(* CODESYS project BProjPLS.export

Project tree, tasks and I/O mapping:
  application Application
    libraries: Util, * (System); WagoAppBuilding, 1.0.2.5 (WAGO); WagoSolMTP, 2.7.0.0 (WAGO); WagoAppMath, 1.1.1.2 (WAGO); WagoAppRTU, 1.2.13.1 (WAGO)
    task PLC_Task (cyclic, interval t#50ms, priority 15) calls PLC_PRG
    task TrendRecordingTask (cyclic, interval 100 ms, priority 15) calls VisuTrendStorageAccess.GlobalInstances.g_TrendRecordingManager.CyclicCall
    global variables GVL
    global variables LVL
    program Binary [ST]
    program Control_System_Analog [ST]
    program Controller [ST]
    program Engine_Control [FBD]: AzimuthThrusters_1, AzimuthThrusters_2, SideThrusters
    program PLC_PRG [ST]
    program Search_Lights [FBD]
    program Tank_Control [FBD]: DieselTank_1, DieselTank_2
    function block Tank_Simulation [FBD]
    program Tempered_Tank [FBD]
    Symbols
  text list GlobalTextList
*)

// Application/GVL
{attribute 'qualified_only'}
VAR_GLOBAL
 	


// Auto pilot
AutoPilot: BOOL; 
iActualDir:INT;
iDestination:INT;
iDirection:INT;
rSTW:REAL;
rCurrent:REAL;
iDepth:INT;
iCurrentDir:INT;




// Main Thrusters
AzimuthPort_Effect: REAL; 
AzimuthPort_Temp: REAL;
AzimuthPort_Angle: REAL;
AzimuthPort_OilPressure: REAL; 

AzimuthStarboard_Effect: REAL; 
AzimuthStarboard_Temp: REAL;
AzimuthStarboard_Angle: REAL;
AzimuthStarboard_OilPressure: REAL; 

// Side Thrusters 
BowThruster_Effect: REAL;
BowThruster_Temp: REAL;
AftThruster_Effect: REAL;
AftThruster_Temp: REAL;

// Diesel Tank
rPump_Tank1: REAL;
rPump_Reserve1: REAL;
Level_Tank1: REAL;
Level_Reserve1: REAL;
Temperature_Tank1: REAL;
Temperature_Reserve1: REAL;

rPump_Tank2: REAL; 
rPump_Reserve2: REAL;
Level_Tank2: REAL;
Level_Reserve2: REAL;
Temperature_Tank2: REAL;
Temperature_Reserve2: REAL;

// Tempered Tank
TemperedTank1_Level:REAL;
TemperedTank1_Temp:REAL;
TemperedTank1_Heat:BOOL;
TemperedTank1_PumpEffect:INT;
TemperedTank1_PumpOn:BOOL;
END_VAR

// Application/LVL
{attribute 'qualified_only'}
VAR_GLOBAL
	

//Controller
iBinary: INT; 
xDI1, xDI2,xDI3,xDI4,xDI5,xDI6: BOOL;
rVoltage:REAL;




END_VAR

// Application/PLC_PRG
PROGRAM PLC_PRG
VAR
END_VAR

Binary();
Control_System_Analog();
Tank_Control();
Engine_Control();
Search_Lights();
Tempered_Tank();
Controller();

END_PROGRAM

// Application/Binary
PROGRAM Binary
VAR
//binary value holders
B1,B2,B3,B4,B5,B6: INT;
	

// flip flop ikke i bruk
flip_flop_1, flip_flop_2, flip_flop_3, flip_flop_4, flip_flop_5,
flip_flop_6, flip_flop_7: fbLatchingRelay;


	
END_VAR

// BINERY switches for button DI1 - DI6, when DI8 is OFF. 	
IF NOT DI8 THEN
	IF DI1 THEN
		B1:=1;
	ELSE
		B1:=0;
	END_IF
	IF DI2 THEN
		B2:=2;
	ELSE
		B2:=0;
	END_IF
	IF DI3 THEN
		B3:=4;
	ELSE
		B3:=0;
	END_IF
	IF DI4 THEN
		B4:=8;
	ELSE
		B4:=0;
	END_IF
	IF DI5 THEN
		B5:=16;
	ELSE
		B5:=0;
	END_IF
	IF DI6 THEN
		B6:=32;
	ELSE
		B6:=0;
	END_IF
	
	LVL.iBinary:=B1+B2+B3+B4+B5+B6;
	
END_IF

// BOOLEAN swithces DI1-DI6 when DI8 is ON
IF DI8 THEN
	flip_flop_1(xButton:=DI1);
	flip_flop_2(xButton:=DI2);
	flip_flop_3(xButton:=DI3);
	flip_flop_4(xButton:=DI4);
	flip_flop_5(xButton:=DI5);
	flip_flop_6(xButton:=DI6);
	flip_flop_7(xButton:=DI7);
	
	
	// test1:=flip_flop_1.xSwitchActuator;
	// test2:=flip_flop_2.xSwitchActuator;
	
	GVL.AutoPilot:=flip_flop_1.xSwitchActuator;
	   
	
END_IF

END_PROGRAM

// Application/Control_System_Analog
PROGRAM Control_System_Analog
VAR
	r_xCurrent:REAL;
	r_yCurrent:REAL;
	iCurrentDirRel:INT;
	rWind:REAL:=3.5;
	iWindDir:INT :=35;
	rsTimer:RS;
	tonTimer:ton;
	rRegulator:REAL;
	Course:AnaView;
	Speed:AnaView;
	
	//Depth
	arrDepth:ARRAY[0..20]OF INT :=[53,57,61,70,71,73,69,60,57,58,55,70,75,74,76,70,65,63,62,59,58];
	i:INT:=0;
	tonDepth:ton;
	rsDepth:RS;
	Depth_View:AnaView;
	
    //Autopilot
	rCOG: REAL;
		
	END_VAR

//Styresystem fart + control
tonTimer(IN:=rsTimer.Q1,PT:=T#1S);
rsTimer(SET:=TRUE,RESET1:=tonTimer.Q);
IF DI7 AND NOT DI8 AND LVL.iBinary<=7 THEN
	rRegulator:=TO_REAL(iwRegulator)/3276.0;
	IF LVL.iBinary= 4 AND tonTimer.Q AND NOT GVL.AutoPilot THEN
		GVL.iDirection:=GVL.iDirection+ (TO_INT(rRegulator)-5); // styres likt med controller for thruster angle  
		IF GVL.iDirection>=360 THEN
			GVL.iDirection:=GVL.iDirection-360;
		ELSIF GVL.iDirection<0 THEN
			GVL.iDirection:=GVL.iDirection+360;
		END_IF
		Course(TagName:='Ship Course',V:=GVL.iDirection,VSclMin:=360,VSclMax:=0,VUnit:=eUnits_IEC61158.degree);
	END_IF
	IF LVL.iBinary=1 AND NOT GVL.AutoPilot THEN 
		GVL.rSTW:=rRegulator*1.032-3.0; // kobles opp mot thruster effekt 
		Speed(TagName:='Ship Speed',V:=GVL.rSTW,VSclMin:=-3,VSclMax:=10,VUnit:=eUnits_IEC61158.knot);
	END_IF
	
END_IF




//Dybdemåler   --- en output skal være global 
rsDepth(SET:=TRUE,RESET1:=tonDepth.Q);
tonDepth(IN:=rsDepth.Q1,PT:=T#2S);
IF tonDepth.Q THEN
		GVL.iDepth:=-arrDepth[i];
		Depth_View(TagName:='Depth',V:=GVL.iDepth);
		i:=i+1;
		IF i=20 THEN 
			i:=0;
		END_IF
	END_IF
	
	
	
//Current
iCurrentDirRel:=GVL.iCurrentDir-GVL.iDirection;
IF iCurrentDirRel>=360 THEN
	iCurrentDirRel:=iCurrentDirRel - 360;
ELSIF iCurrentDirRel <0 THEN
	iCurrentDirRel := iCurrentDirRel + 360;
END_IF
IF GVL.rCurrent<GVL.rSTW THEN 
r_xCurrent:=-(cos_r(degreeToAngle(iCurrentDirRel))*GVL.rCurrent);//legg til speed heading
r_yCurrent:=-(sin_r(degreeToAngle(iCurrentDirRel))*GVL.rCurrent); 
rCOG:=sqrt_l(((GVL.rSTW+r_xCurrent)*(GVL.rSTW+r_xCurrent))+((r_yCurrent)*(r_yCurrent)));
GVL.iActualDir:=TO_INT(angleToDegree_r(arcTan(r_yCurrent/(GVL.rSTW+r_xCurrent)))+GVL.iDirection);
IF rCOG=0 THEN GVL.iActualDir:=GVL.iDirection; END_IF
IF GVL.iActualDir<0 THEN GVL.iActualDir:=GVL.iActualDir+360; ELSIF GVL.iActualDir>=360 THEN GVL.iActualDir:=GVL.iActualDir-360; END_IF
	
END_IF





//AutoPilot
IF GVL.AutoPilot THEN
	IF GVL.iDestination=GVL.iActualDir THEN GVL.BowThruster_Effect:=0;GVL.AzimuthPort_Angle:=0;GVL.AzimuthStarboard_Angle:=0;END_IF
	IF GVL.iActualDir<0 THEN GVL.iActualDir:=GVL.iActualDir+360; ELSIF GVL.iActualDir>=360 THEN GVL.iActualDir:=GVL.iActualDir-360; END_IF
	IF GVL.iDirection<0 THEN GVL.iDirection:=GVL.iDirection+360; ELSIF GVL.iDirection>=360 THEN GVL.iDirection:=GVL.iDirection-360; END_IF
	IF GVL.iActualDir>GVL.iDestination AND tontimer.Q THEN
		IF GVL.iActualDir-GVL.iDestination>180 THEN // checks if course minus destination is greater than 180 degrees 
			
			IF GVL.iActualDir-GVL.iDestination>340 THEN // 
				GVL.iDirection:=GVL.iDirection+3;
				GVL.BowThruster_Effect := 100;   //autopilot side and main engines
				GVL.AzimuthPort_Angle := 35;
				GVL.AzimuthStarboard_Angle := 35;
			
			ELSIF GVL.iActualDir-GVL.iDestination>350 THEN
				GVL.iDirection:=GVL.iDirection+2;
				GVL.BowThruster_Effect := 50;   //autopilot side and main engines
				GVL.AzimuthPort_Angle := 20;
				GVL.AzimuthStarboard_Angle := 20;
			ELSE 
				GVL.iDirection:=GVL.iDirection+1;
				GVL.BowThruster_Effect := 25;   //autopilot side and main engines
				GVL.AzimuthPort_Angle := 10;
				GVL.AzimuthStarboard_Angle := 10;
			END_IF
		ELSE
		
			IF GVL.iActualDir-GVL.iDestination>20 THEN
			GVL.iDirection:=GVL.iDirection-3;
			
				GVL.BowThruster_Effect := -100;   //autopilot side and main engines
				GVL.AzimuthPort_Angle := -35;
				GVL.AzimuthStarboard_Angle := -35;
			ELSIF GVL.iDestination-GVL.iActualDir>10 THEN
				GVL.iDirection:=GVL.iDirection-2;
					GVL.BowThruster_Effect := -50;   //autopilot side and main engines
				GVL.AzimuthPort_Angle := -20;
				GVL.AzimuthStarboard_Angle := -20;
			ELSE
				GVL.iDirection:=GVL.iDirection-1;
					GVL.BowThruster_Effect := -25;   //autopilot side and main engines
				GVL.AzimuthPort_Angle := -10;
				GVL.AzimuthStarboard_Angle := -10;
			END_IF
		END_IF
	ELSIF GVL.iDestination>GVL.iActualDir AND tonTimer.Q THEN
		IF GVL.iDestination-GVL.iActualDir>180 THEN
			IF GVL.iDestination-GVL.iActualDir>340 THEN
				GVL.iDirection:=GVL.iDirection-3;
					GVL.BowThruster_Effect := -100;   //autopilot side and main engines
				GVL.AzimuthPort_Angle := -35;
				GVL.AzimuthStarboard_Angle := -35;
			ELSIF GVL.iDestination-GVL.iActualDir>350 THEN
				GVL.iDirection:=GVL.iDirection-2;
					GVL.BowThruster_Effect := -50;   //autopilot side and main engines
				GVL.AzimuthPort_Angle := -20;
				GVL.AzimuthStarboard_Angle := -20;
				
			ELSE
				GVL.iDirection:=GVL.iDirection-1;
					GVL.BowThruster_Effect := -25;   //autopilot side and main engines
				GVL.AzimuthPort_Angle := -10;
				GVL.AzimuthStarboard_Angle := -10;
			END_IF
		ELSE
			IF GVL.iDestination-GVL.iActualDir>20 THEN
				GVL.iDirection:=GVL.iDirection+3;
					GVL.BowThruster_Effect := 100;   //autopilot side and main engines
				GVL.AzimuthPort_Angle := 35;
				GVL.AzimuthStarboard_Angle := 35;
			ELSIF GVL.iDestination-GVL.iActualDir>10 THEN
				GVL.iDirection:=GVL.iDirection+2;
					GVL.BowThruster_Effect := 50;   //autopilot side and main engines
				GVL.AzimuthPort_Angle := 20;
				GVL.AzimuthStarboard_Angle := 20;
			ELSE
				GVL.iDirection:=GVL.iDirection+1;
					GVL.BowThruster_Effect := 25;   //autopilot side and main engines
				GVL.AzimuthPort_Angle := 10;
				GVL.AzimuthStarboard_Angle := 10;
			END_IF
		END_IF
	END_IF
END_IF

END_PROGRAM

// Application/Controller
PROGRAM Controller
VAR
tonTimer: ton; 
rsTimer: rs; 	
rRegulator: REAL;



END_VAR


// Direction
tonTimer(IN:=rsTimer.Q1,PT:=T#1S);
rsTimer(SET:=TRUE,RESET1:=tonTimer.Q);



 
 
 //Scales regulator signal
  rRegulator := FU2POINT(IoConfig_Globals_Mapping.iwRegulator,0,0,32760,100); 
  
 
 IF DI7 AND NOT DI8 AND tonTimer.Q THEN  
     LVL.rVoltage:=TO_REAL(TO_INT(rRegulator))/10;
   
      //Azimuth Thrusters 

     IF LVL.iBinary= 1 THEN 
        GVL.AzimuthPort_Effect:=FU2POINT(LVL.rVoltage,0,-30,10,100);
		GVL.AzimuthStarboard_Effect:=FU2POINT(LVL.rVoltage,0,-30,10,100);
     ELSIF LVL.iBinary= 2 THEN  
           GVL.AzimuthPort_Temp:=FU2POINT(LVL.rVoltage,0,0,10,200);
		   GVL.AzimuthStarboard_Temp:=FU2POINT(LVL.rVoltage,0,0,10,200);
     ELSIF LVL.iBinary= 4 AND NOT GVL.autopilot THEN 
           GVL.AzimuthPort_Angle:=FU2POINT(LVL.rVoltage,0,-35,10,35);
		   GVL.AzimuthStarboard_Angle:=FU2POINT(LVL.rVoltage,0,-35,10,35);
     ELSIF LVL.iBinary= 8 THEN 
           GVL.AzimuthPort_OilPressure:=FU2POINT(LVL.rVoltage,0,0,10,100);
		   GVL.AZIMUTHSTARBOARD_OILPRESSURE:=FU2POINT(LVL.RVOLTAGE,0,0,10,100);

     //Side Thrusters. 
	  ELSIF LVL.iBinary=16+1 AND NOT GVL.autopilot THEN  
            GVL.BowThruster_Effect:=FU2POINT(LVL.rVoltage,0,-100,10,100);
	  ELSIF LVL.iBinary=16+2 
         THEN  GVL.BowThruster_Temp:=FU2POINT(LVL.rVoltage,0,-10,10,200);
   
      ELSIF LVL.iBinary=16+4 
         THEN  GVL.AftThruster_Effect:=FU2POINT(LVL.rVoltage,0,-100,10,100);
      ELSIF LVL.iBinary=16+8
         THEN  GVL.AftThruster_Temp:=FU2POINT(LVL.rVoltage,0,-10,10,200);
		
    // Diesel Tanks 
	ELSIF LVL.iBinary=32+1 THEN
		GVL.Level_Tank1:=FU2POINT(LVL.rVoltage,0,0,10,200);
		GVL.Level_Tank2:=FU2POINT(LVL.rVoltage,0,0,10,200);
	ELSIF LVL.iBinary=32+2 THEN
		GVL.Level_Reserve1:=FU2POINT(LVL.rVoltage,0,0,10,50);
		GVL.Level_Reserve2:=FU2POINT(LVL.rVoltage,0,0,10,50);
	ELSIF LVL.iBinary=32+4 THEN
		GVL.Temperature_Tank1:=FU2POINT(LVL.rVoltage,0,0,10,225);
		GVL.Temperature_Tank2:=FU2POINT(LVL.rVoltage,0,0,10,225);
	ELSIF LVL.iBinary=32+8 THEN
		GVL.Temperature_Reserve1:=FU2POINT(LVL.rVoltage,0,0,10,225);
		GVL.Temperature_Reserve2:=FU2POINT(LVL.rVoltage,0,0,10,225);
	END_IF
			 
   
         
	
END_IF

END_PROGRAM

// Application/Tank_Control
PROGRAM Tank_Control
VAR	
// Variables for fuel controll	
Engine_Effect1: REAL;
Fuelusage1: REAL;

Engine_Effect2: REAL;
Fuelusage2: REAL;


	//Diesel Tank 1

	
	Level_Tank1_Mon: AnaMon :=(VTHLim:=200,VALLim:=1,VWLLim:=10,V:=50);
	Level_Reserve1_Mon: AnaMon :=(VTHLim:=50,VALLim:=1,VWLLim:=5);
	Temperature_Tank1_Mon: AnaMon :=(VAHLim:=200,VWHLim:=100);
	Temperature_Reserve1_Mon: AnaMon :=(VAHLim:=200,VWHLim:=100);



	Pump_Tank1_View: AnaView;
	Pump_Reserve1_View: AnaView;
	

    //Diesel Tank 2


	
	Pump_Tank2_View: AnaView;
	Pump_Reserve2_View: AnaView;
	Level_Tank2_Mon: AnaMon :=(VTHLim:=200,VALLim:=1,VWLLim:=10);
	Level_Reserve2_Mon: AnaMon :=(VTHLim:=50,VALLim:=1,VWLLim:=5);
	Temperature_Tank2_Mon: AnaMon :=(VAHLim:=200,VWHLim:=100);
	Temperature_Reserve2_Mon: AnaMon :=(VAHLim:=200,VWHLim:=100);

	
END_VAR
VAR // added by the converter: edge detectors and wires of the graphical bodies
    _w1, _w2, _w3, _w4 : BOOL;
END_VAR

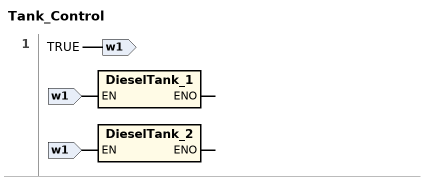
// NETWORK 1
DieselTank_1();
DieselTank_2();

ACTION DieselTank_1:
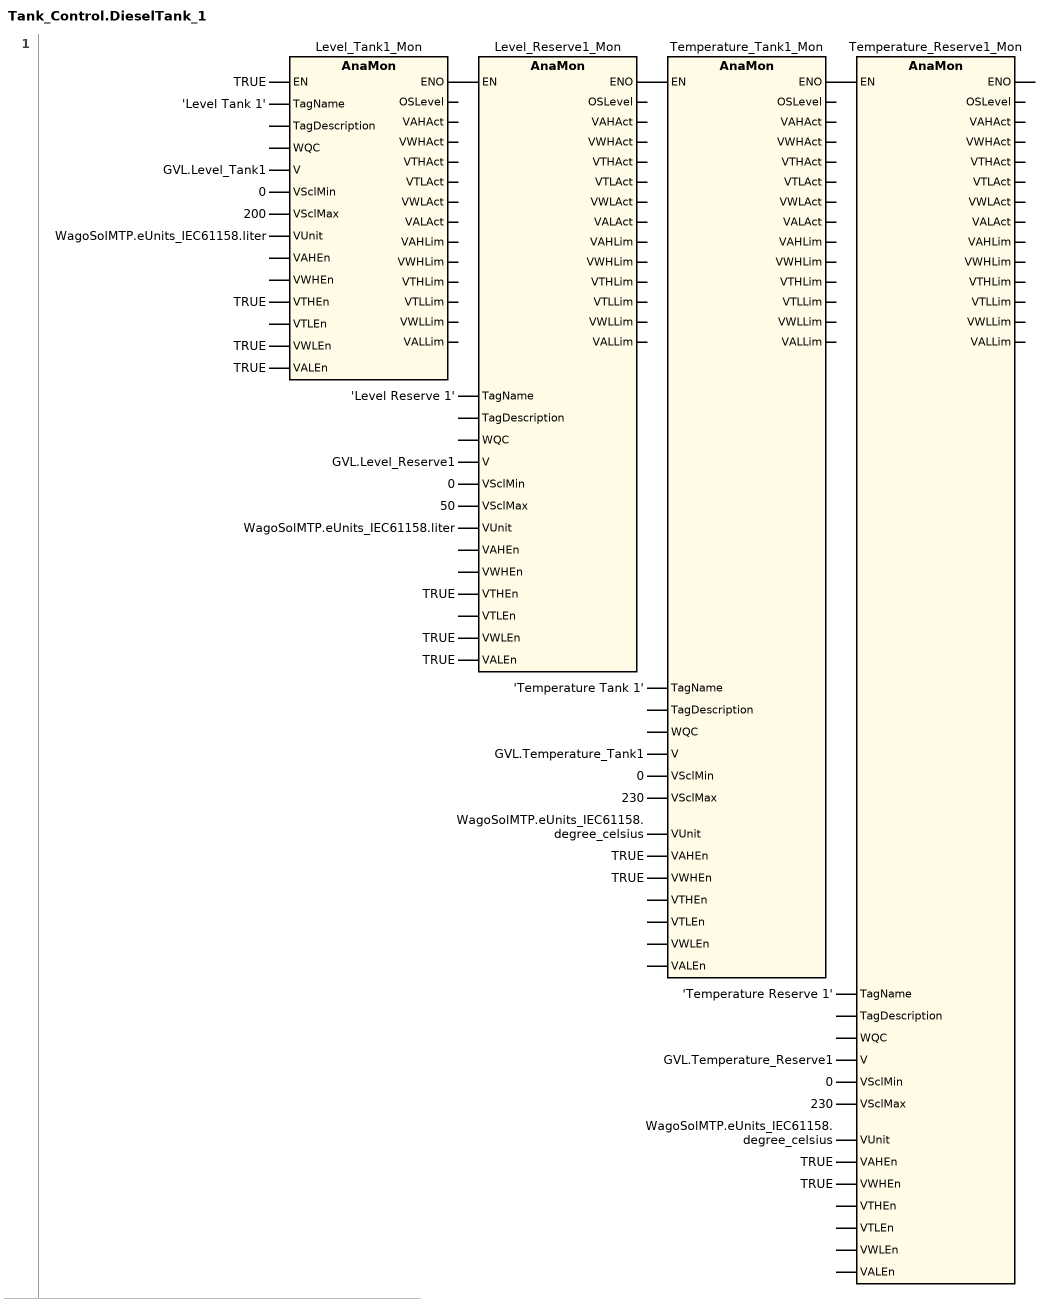
// NETWORK 1
Level_Tank1_Mon(
    TagName := 'Level Tank 1',
    V := GVL.Level_Tank1,
    VSclMin := 0,
    VSclMax := 200,
    VUnit := WagoSolMTP.eUnits_IEC61158.liter,
    VTHEn := TRUE,
    VWLEn := TRUE,
    VALEn := TRUE); // AnaMon
Level_Reserve1_Mon(
    TagName := 'Level Reserve 1',
    V := GVL.Level_Reserve1,
    VSclMin := 0,
    VSclMax := 50,
    VUnit := WagoSolMTP.eUnits_IEC61158.liter,
    VTHEn := TRUE,
    VWLEn := TRUE,
    VALEn := TRUE); // AnaMon
Temperature_Tank1_Mon(
    TagName := 'Temperature Tank 1',
    V := GVL.Temperature_Tank1,
    VSclMin := 0,
    VSclMax := 230,
    VUnit := WagoSolMTP.eUnits_IEC61158.degree_celsius,
    VAHEn := TRUE,
    VWHEn := TRUE); // AnaMon
Temperature_Reserve1_Mon(
    TagName := 'Temperature Reserve 1',
    V := GVL.Temperature_Reserve1,
    VSclMin := 0,
    VSclMax := 230,
    VUnit := WagoSolMTP.eUnits_IEC61158.degree_celsius,
    VAHEn := TRUE,
    VWHEn := TRUE); // AnaMon

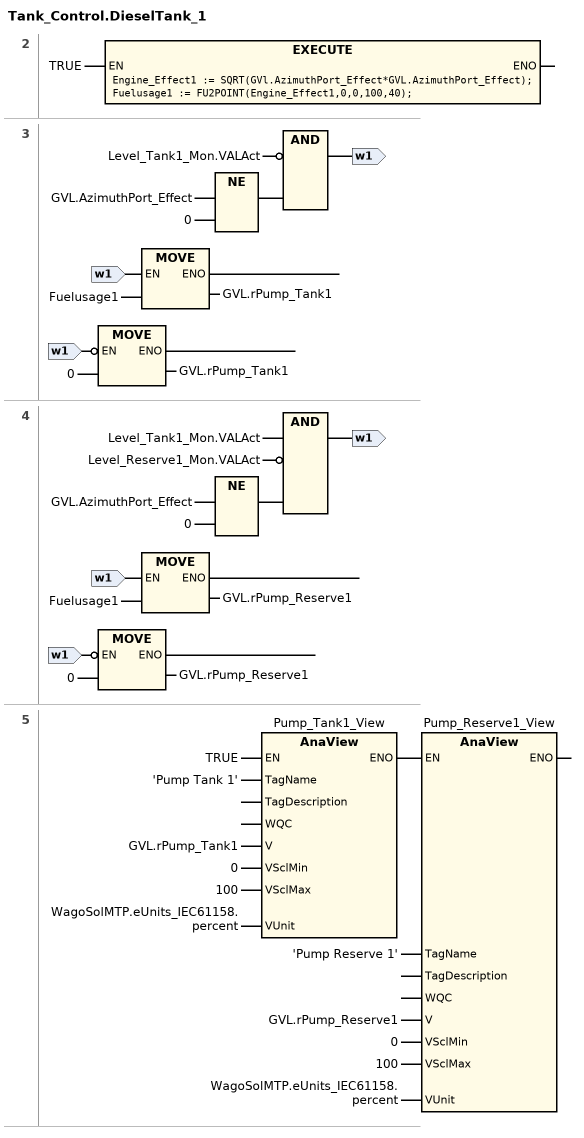
// NETWORK 2
Engine_Effect1 := SQRT(GVl.AzimuthPort_Effect*GVL.AzimuthPort_Effect);
Fuelusage1 := FU2POINT(Engine_Effect1,0,0,100,40);

// NETWORK 3
_w1 := NOT Level_Tank1_Mon.VALAct AND GVL.AzimuthPort_Effect <> 0;
IF _w1 THEN GVL.rPump_Tank1 := Fuelusage1; END_IF
IF NOT _w1 THEN GVL.rPump_Tank1 := 0; END_IF

// NETWORK 4
_w2 := Level_Tank1_Mon.VALAct AND NOT Level_Reserve1_Mon.VALAct AND GVL.AzimuthPort_Effect <> 0;
IF _w2 THEN GVL.rPump_Reserve1 := Fuelusage1; END_IF
IF NOT _w2 THEN GVL.rPump_Reserve1 := 0; END_IF

// NETWORK 5
Pump_Tank1_View(
    TagName := 'Pump Tank 1',
    V := GVL.rPump_Tank1,
    VSclMin := 0,
    VSclMax := 100,
    VUnit := WagoSolMTP.eUnits_IEC61158.percent); // AnaView
Pump_Reserve1_View(
    TagName := 'Pump Reserve 1',
    V := GVL.rPump_Reserve1,
    VSclMin := 0,
    VSclMax := 100,
    VUnit := WagoSolMTP.eUnits_IEC61158.percent); // AnaView
END_ACTION

ACTION DieselTank_2:
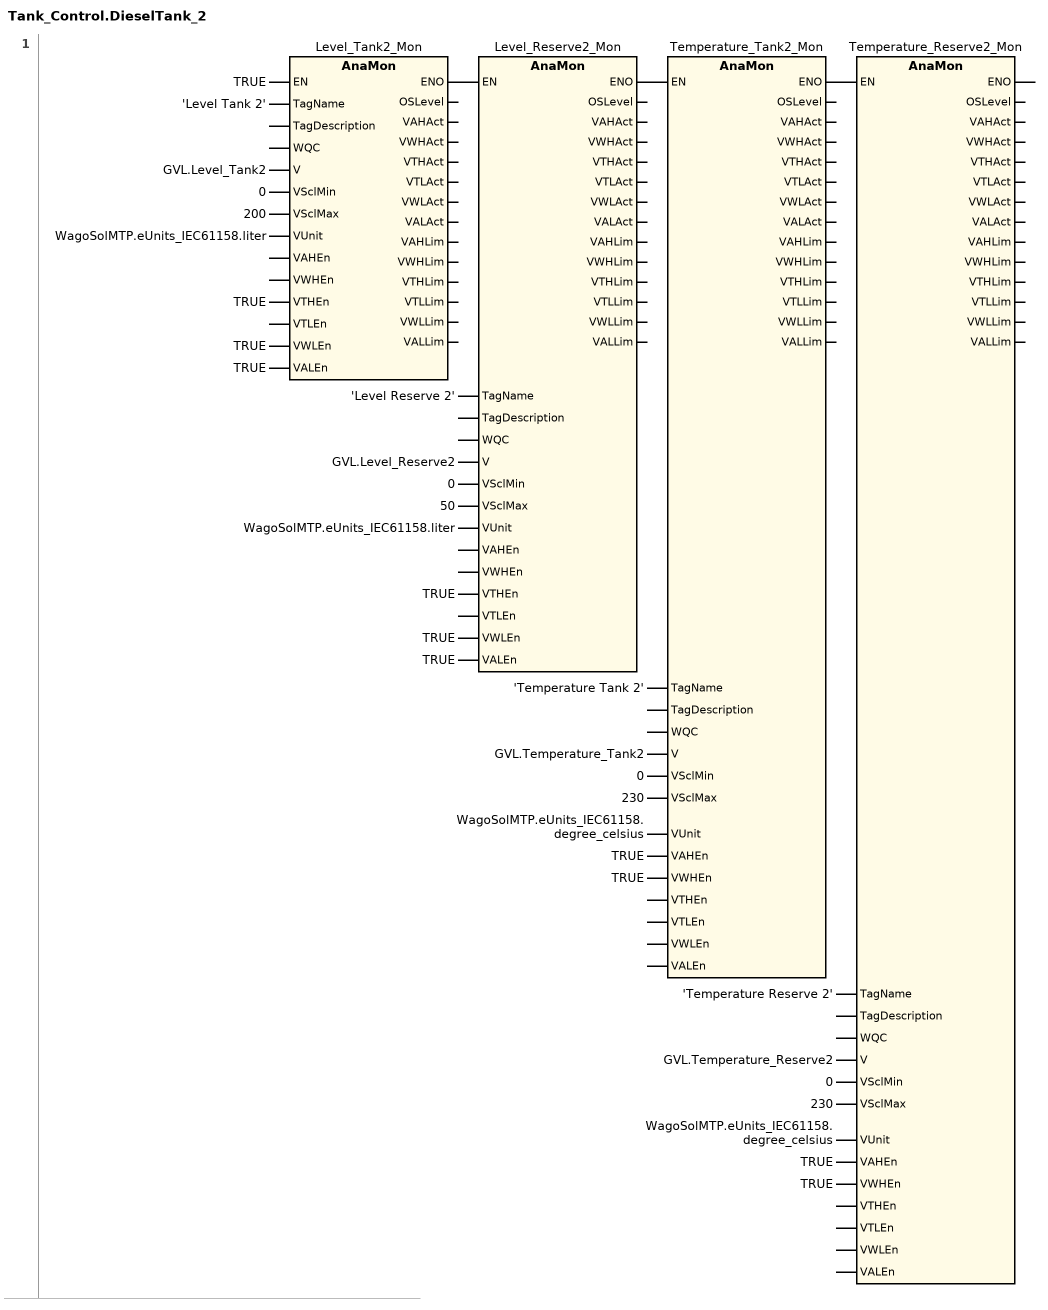
// NETWORK 1
Level_Tank2_Mon(
    TagName := 'Level Tank 2',
    V := GVL.Level_Tank2,
    VSclMin := 0,
    VSclMax := 200,
    VUnit := WagoSolMTP.eUnits_IEC61158.liter,
    VTHEn := TRUE,
    VWLEn := TRUE,
    VALEn := TRUE); // AnaMon
Level_Reserve2_Mon(
    TagName := 'Level Reserve 2',
    V := GVL.Level_Reserve2,
    VSclMin := 0,
    VSclMax := 50,
    VUnit := WagoSolMTP.eUnits_IEC61158.liter,
    VTHEn := TRUE,
    VWLEn := TRUE,
    VALEn := TRUE); // AnaMon
Temperature_Tank2_Mon(
    TagName := 'Temperature Tank 2',
    V := GVL.Temperature_Tank2,
    VSclMin := 0,
    VSclMax := 230,
    VUnit := WagoSolMTP.eUnits_IEC61158.degree_celsius,
    VAHEn := TRUE,
    VWHEn := TRUE); // AnaMon
Temperature_Reserve2_Mon(
    TagName := 'Temperature Reserve 2',
    V := GVL.Temperature_Reserve2,
    VSclMin := 0,
    VSclMax := 230,
    VUnit := WagoSolMTP.eUnits_IEC61158.degree_celsius,
    VAHEn := TRUE,
    VWHEn := TRUE); // AnaMon

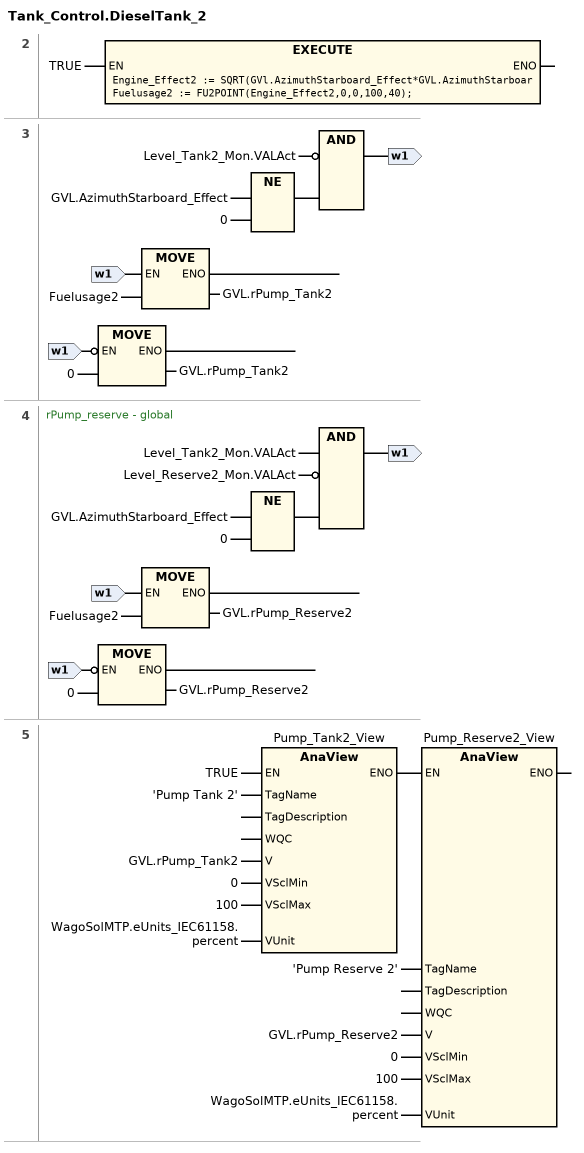
// NETWORK 2
Engine_Effect2 := SQRT(GVl.AzimuthStarboard_Effect*GVL.AzimuthStarboard_Effect);
Fuelusage2 := FU2POINT(Engine_Effect2,0,0,100,40);

// NETWORK 3
_w3 := NOT Level_Tank2_Mon.VALAct AND GVL.AzimuthStarboard_Effect <> 0;
IF _w3 THEN GVL.rPump_Tank2 := Fuelusage2; END_IF
IF NOT _w3 THEN GVL.rPump_Tank2 := 0; END_IF

// NETWORK 4
// rPump_reserve - global
_w4 := Level_Tank2_Mon.VALAct AND NOT Level_Reserve2_Mon.VALAct AND GVL.AzimuthStarboard_Effect <> 0;
IF _w4 THEN GVL.rPump_Reserve2 := Fuelusage2; END_IF
IF NOT _w4 THEN GVL.rPump_Reserve2 := 0; END_IF

// NETWORK 5
Pump_Tank2_View(
    TagName := 'Pump Tank 2',
    V := GVL.rPump_Tank2,
    VSclMin := 0,
    VSclMax := 100,
    VUnit := WagoSolMTP.eUnits_IEC61158.percent); // AnaView
Pump_Reserve2_View(
    TagName := 'Pump Reserve 2',
    V := GVL.rPump_Reserve2,
    VSclMin := 0,
    VSclMax := 100,
    VUnit := WagoSolMTP.eUnits_IEC61158.percent); // AnaView
END_ACTION

END_PROGRAM

// Application/Engine_Control
PROGRAM Engine_Control
VAR


    //AzimuthThruster
   
 
    //Side Thrusters
   
	
	//Thruster 1
	AzimuthPort_Angle_View: AnaView;
	AzimuthPort_OilPressure_View: AnaView;
	
	AzimuthPort_Temp_Mon: AnaMon:= (VAHLim:= 200, VWHLim:= 150, VALLim:=-10);
	AzimuthPort_Effect_Mon: AnaMon:= (VAHLim:= 100, VTHLim:=80, VALLim:= -30);
	
	
	
	//Thruster 2
	AzimuthStarboard_Angle_View: AnaView;
	AzimuthStarboard_OilPressure_View: AnaView;
	
	AzimuthStarboard_Temp_Mon: AnaMon:= (VAHLim:= 200, VWHLim:= 150, VALLim:=-10);
	AzimuthStarboard_Effect_Mon: AnaMon:= (VAHLim:= 100, VTHLim:=80, VALLim:= -30);
	
	
	
	// Bow Thruster 1
    
    BowThruster1_Effect_View: AnaView;
	BowThruster1_Temp_View: AnaView;
    
    BowThruster1_Temp_Mon: AnaMon:= (VAHLim:= 200, VWHLim:= 150, VALLim:=-10);
							
	//Bow Thruster 2
   	BowThruster2_Effect_View: AnaView;
	BowThruster2_Temp_View: AnaView;
	
    BowThruster2_Temp_Mon: AnaMon :=(VAHLim:= 200, VWHLim:= 150, VALLim:=-10);
	
	//AftThruster 2 
	AftThruster_Effect_View: AnaView;
	AftThruster_Temp_View: AnaView;
	
    AftThruster_Temp_Mon: AnaMon := (VAHLim:= 200, VWHLim:= 150, VALLim:=-10);
	
	
	
	
 



END_VAR

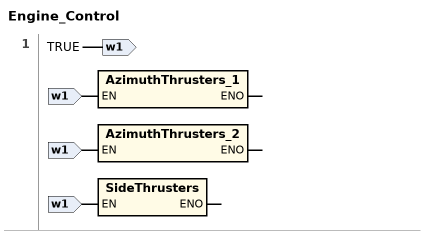
// NETWORK 1
AzimuthThrusters_1();
AzimuthThrusters_2();
SideThrusters();

ACTION AzimuthThrusters_1:
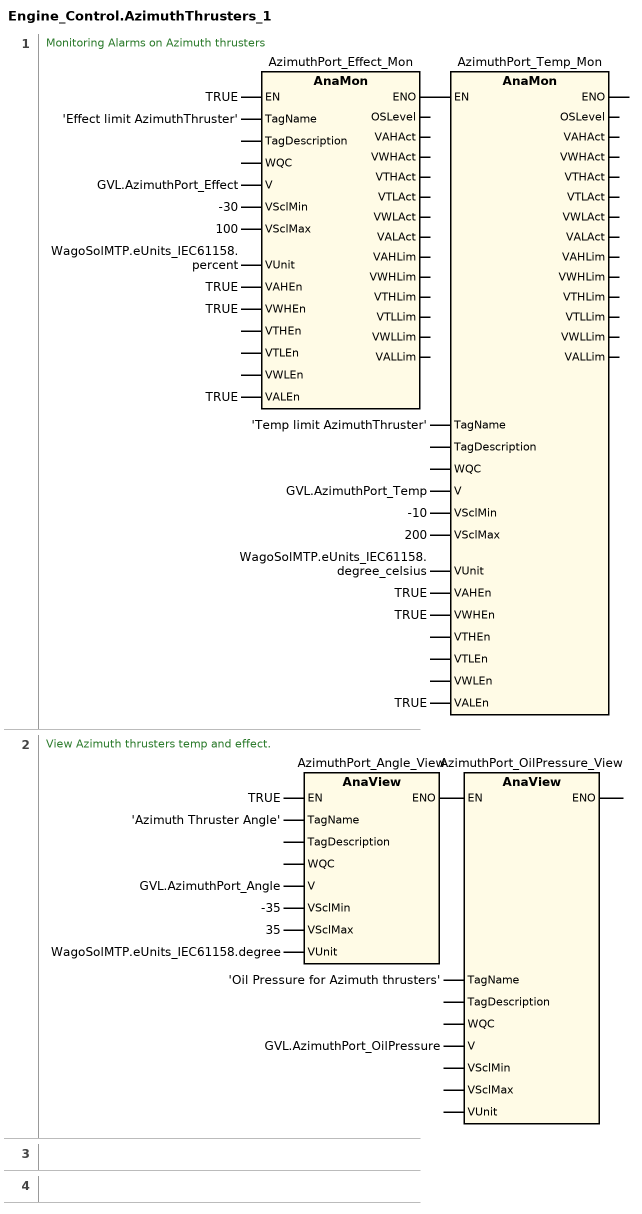
// NETWORK 1
// Monitoring Alarms on Azimuth thrusters
AzimuthPort_Effect_Mon(
    TagName := 'Effect limit AzimuthThruster',
    V := GVL.AzimuthPort_Effect,
    VSclMin := -30,
    VSclMax := 100,
    VUnit := WagoSolMTP.eUnits_IEC61158.percent,
    VAHEn := TRUE,
    VWHEn := TRUE,
    VALEn := TRUE); // AnaMon
AzimuthPort_Temp_Mon(
    TagName := 'Temp limit AzimuthThruster',
    V := GVL.AzimuthPort_Temp,
    VSclMin := -10,
    VSclMax := 200,
    VUnit := WagoSolMTP.eUnits_IEC61158.degree_celsius,
    VAHEn := TRUE,
    VWHEn := TRUE,
    VALEn := TRUE); // AnaMon

// NETWORK 2
// View Azimuth thrusters temp and effect.
AzimuthPort_Angle_View(
    TagName := 'Azimuth Thruster Angle',
    V := GVL.AzimuthPort_Angle,
    VSclMin := -35,
    VSclMax := 35,
    VUnit := WagoSolMTP.eUnits_IEC61158.degree); // AnaView
AzimuthPort_OilPressure_View(TagName := 'Oil Pressure for Azimuth thrusters', V := GVL.AzimuthPort_OilPressure); // AnaView

// NETWORK 3

// NETWORK 4
END_ACTION

ACTION AzimuthThrusters_2:
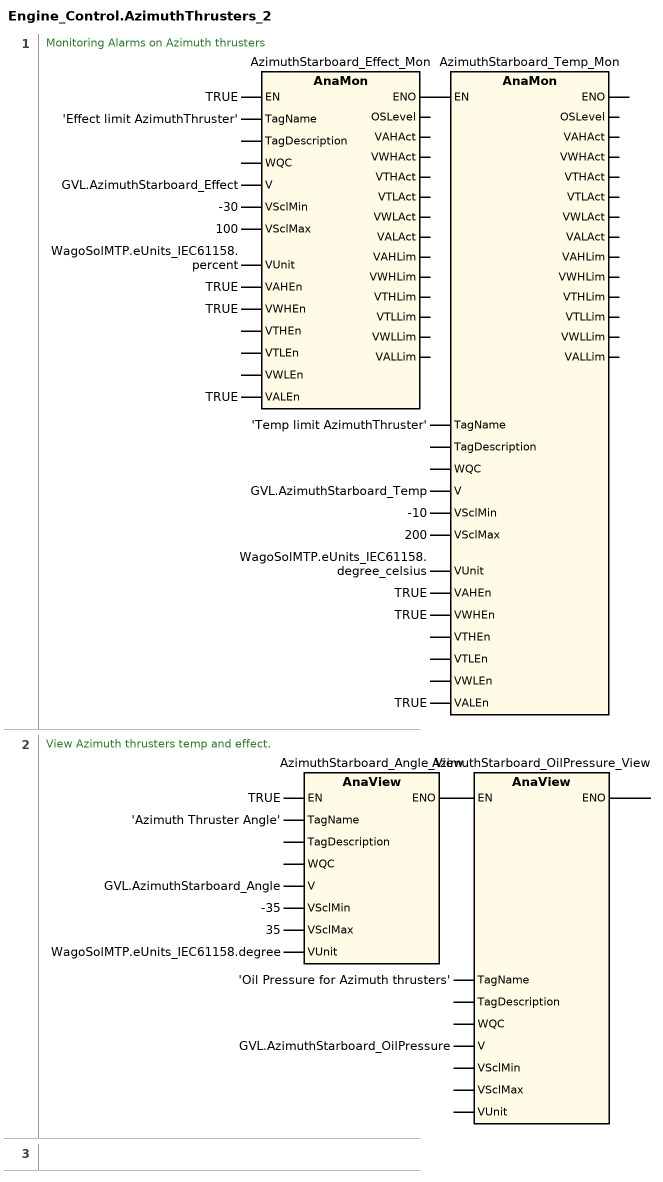
// NETWORK 1
// Monitoring Alarms on Azimuth thrusters
AzimuthStarboard_Effect_Mon(
    TagName := 'Effect limit AzimuthThruster',
    V := GVL.AzimuthStarboard_Effect,
    VSclMin := -30,
    VSclMax := 100,
    VUnit := WagoSolMTP.eUnits_IEC61158.percent,
    VAHEn := TRUE,
    VWHEn := TRUE,
    VALEn := TRUE); // AnaMon
AzimuthStarboard_Temp_Mon(
    TagName := 'Temp limit AzimuthThruster',
    V := GVL.AzimuthStarboard_Temp,
    VSclMin := -10,
    VSclMax := 200,
    VUnit := WagoSolMTP.eUnits_IEC61158.degree_celsius,
    VAHEn := TRUE,
    VWHEn := TRUE,
    VALEn := TRUE); // AnaMon

// NETWORK 2
// View Azimuth thrusters temp and effect.
AzimuthStarboard_Angle_View(
    TagName := 'Azimuth Thruster Angle',
    V := GVL.AzimuthStarboard_Angle,
    VSclMin := -35,
    VSclMax := 35,
    VUnit := WagoSolMTP.eUnits_IEC61158.degree); // AnaView
AzimuthStarboard_OilPressure_View(TagName := 'Oil Pressure for Azimuth thrusters', V := GVL.AzimuthStarboard_OilPressure); // AnaView

// NETWORK 3
END_ACTION

ACTION SideThrusters:
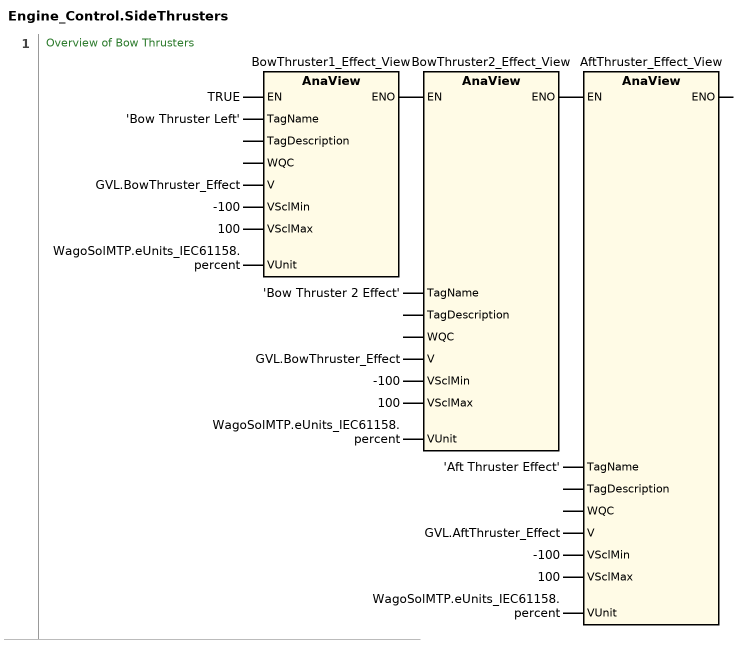
// NETWORK 1
// Overview of Bow Thrusters
BowThruster1_Effect_View(
    TagName := 'Bow Thruster Left',
    V := GVL.BowThruster_Effect,
    VSclMin := -100,
    VSclMax := 100,
    VUnit := WagoSolMTP.eUnits_IEC61158.percent); // AnaView
BowThruster2_Effect_View(
    TagName := 'Bow Thruster 2 Effect',
    V := GVL.BowThruster_Effect,
    VSclMin := -100,
    VSclMax := 100,
    VUnit := WagoSolMTP.eUnits_IEC61158.percent); // AnaView
AftThruster_Effect_View(
    TagName := 'Aft Thruster Effect',
    V := GVL.AftThruster_Effect,
    VSclMin := -100,
    VSclMax := 100,
    VUnit := WagoSolMTP.eUnits_IEC61158.percent); // AnaView

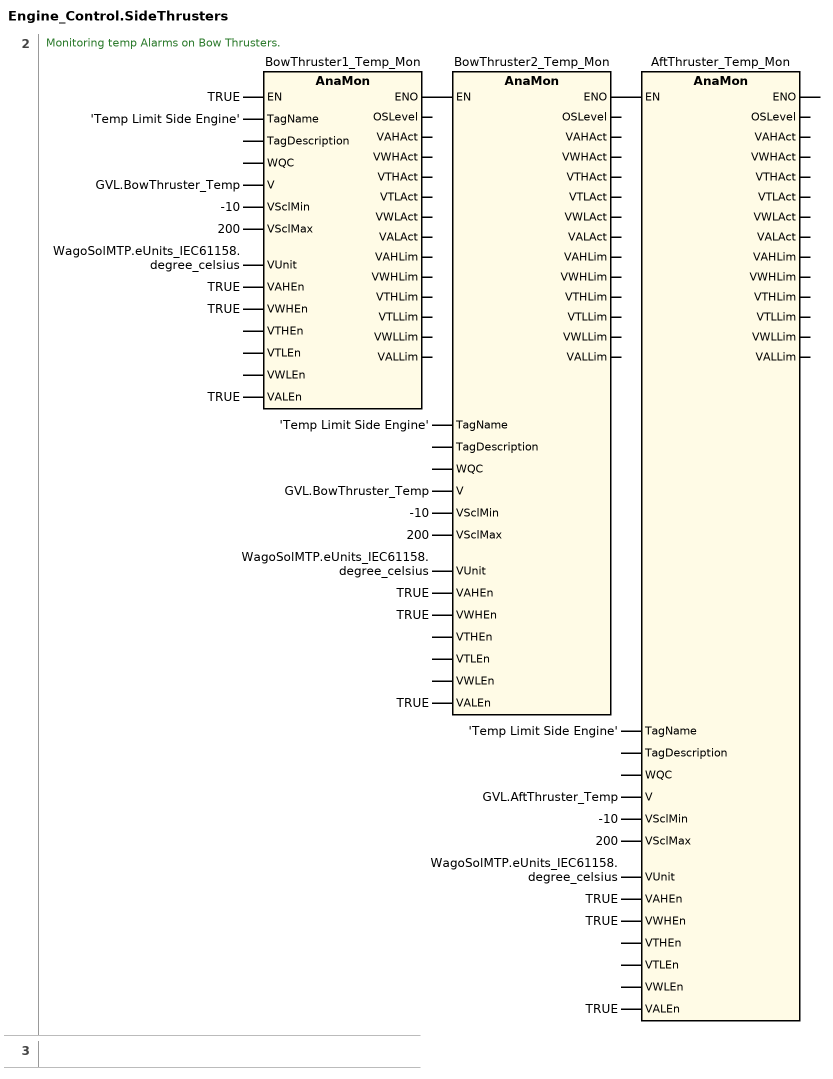
// NETWORK 2
// Monitoring temp Alarms on Bow Thrusters.
BowThruster1_Temp_Mon(
    TagName := 'Temp Limit Side Engine',
    V := GVL.BowThruster_Temp,
    VSclMin := -10,
    VSclMax := 200,
    VUnit := WagoSolMTP.eUnits_IEC61158.degree_celsius,
    VAHEn := TRUE,
    VWHEn := TRUE,
    VALEn := TRUE); // AnaMon
BowThruster2_Temp_Mon(
    TagName := 'Temp Limit Side Engine',
    V := GVL.BowThruster_Temp,
    VSclMin := -10,
    VSclMax := 200,
    VUnit := WagoSolMTP.eUnits_IEC61158.degree_celsius,
    VAHEn := TRUE,
    VWHEn := TRUE,
    VALEn := TRUE); // AnaMon
AftThruster_Temp_Mon(
    TagName := 'Temp Limit Side Engine',
    V := GVL.AftThruster_Temp,
    VSclMin := -10,
    VSclMax := 200,
    VUnit := WagoSolMTP.eUnits_IEC61158.degree_celsius,
    VAHEn := TRUE,
    VWHEn := TRUE,
    VALEn := TRUE); // AnaMon

// NETWORK 3
END_ACTION

END_PROGRAM

// Application/Search_Lights
PROGRAM Search_Lights
VAR
	Search_Light_1: AnaMan;
	Search_Light_2: AnaMan;
	Search_Light_3: AnaMan;
	Search_Light_4: AnaMan;
	Search_Light_5: AnaMan;
	Search_Light_6: AnaMan;
	Search_Light_7: AnaMan;
	Light_Switch_1: BinMan;
	Light_Switch_2: BinMan;
	Light_Switch_3: BinMan;
	Light_Switch_4: BinMan;
	Light_Switch_5: BinMan;
	Light_Switch_6: BinMan;
	Light_Switch_7: BinMan;
END_VAR

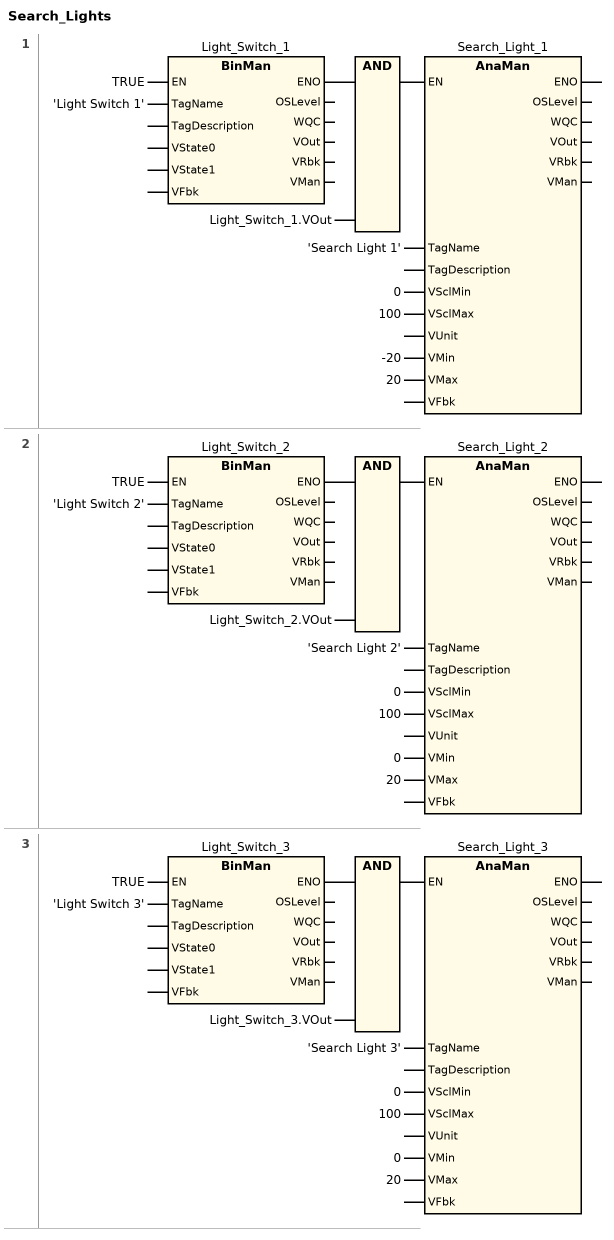
// NETWORK 1
Light_Switch_1(TagName := 'Light Switch 1'); // BinMan
IF TRUE AND Light_Switch_1.VOut THEN
    Search_Light_1(TagName := 'Search Light 1', VSclMin := 0, VSclMax := 100, VMin := -20, VMax := 20); // AnaMan
END_IF

// NETWORK 2
Light_Switch_2(TagName := 'Light Switch 2'); // BinMan
IF TRUE AND Light_Switch_2.VOut THEN
    Search_Light_2(TagName := 'Search Light 2', VSclMin := 0, VSclMax := 100, VMin := 0, VMax := 20); // AnaMan
END_IF

// NETWORK 3
Light_Switch_3(TagName := 'Light Switch 3'); // BinMan
IF TRUE AND Light_Switch_3.VOut THEN
    Search_Light_3(TagName := 'Search Light 3', VSclMin := 0, VSclMax := 100, VMin := 0, VMax := 20); // AnaMan
END_IF

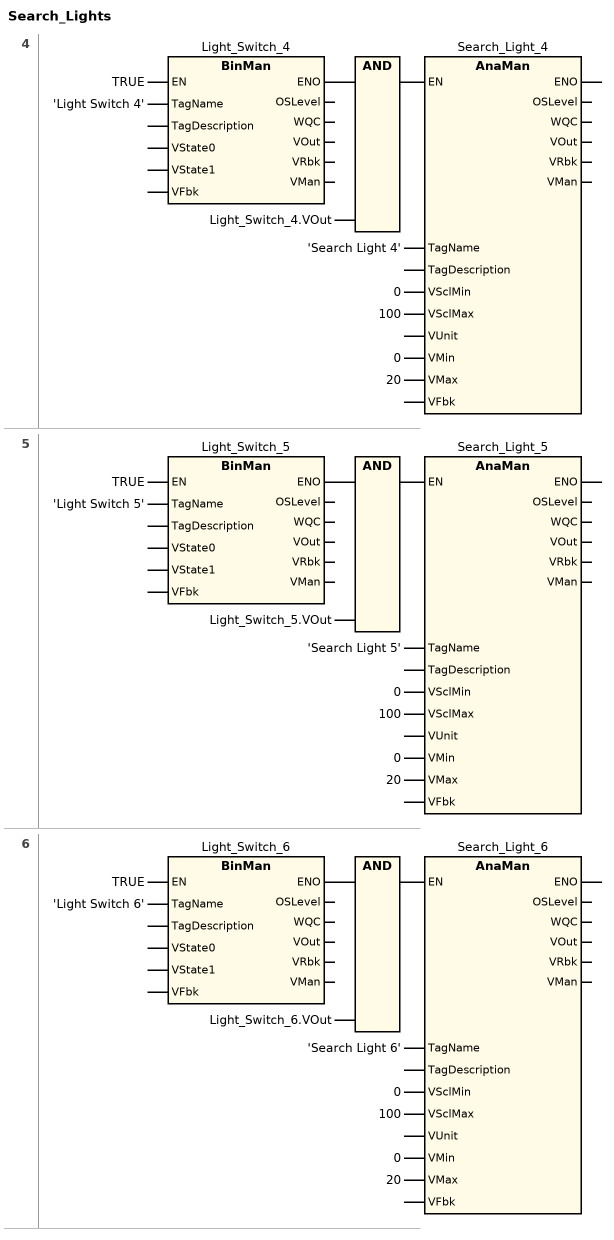
// NETWORK 4
Light_Switch_4(TagName := 'Light Switch 4'); // BinMan
IF TRUE AND Light_Switch_4.VOut THEN
    Search_Light_4(TagName := 'Search Light 4', VSclMin := 0, VSclMax := 100, VMin := 0, VMax := 20); // AnaMan
END_IF

// NETWORK 5
Light_Switch_5(TagName := 'Light Switch 5'); // BinMan
IF TRUE AND Light_Switch_5.VOut THEN
    Search_Light_5(TagName := 'Search Light 5', VSclMin := 0, VSclMax := 100, VMin := 0, VMax := 20); // AnaMan
END_IF

// NETWORK 6
Light_Switch_6(TagName := 'Light Switch 6'); // BinMan
IF TRUE AND Light_Switch_6.VOut THEN
    Search_Light_6(TagName := 'Search Light 6', VSclMin := 0, VSclMax := 100, VMin := 0, VMax := 20); // AnaMan
END_IF

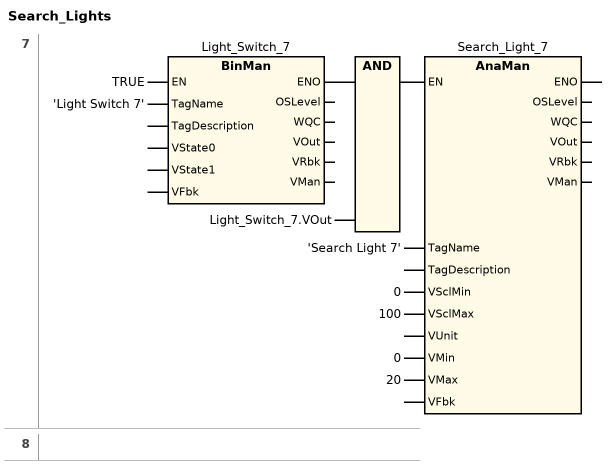
// NETWORK 7
Light_Switch_7(TagName := 'Light Switch 7'); // BinMan
IF TRUE AND Light_Switch_7.VOut THEN
    Search_Light_7(TagName := 'Search Light 7', VSclMin := 0, VSclMax := 100, VMin := 0, VMax := 20); // AnaMan
END_IF

// NETWORK 8

END_PROGRAM

// Application/Tempered_Tank
PROGRAM Tempered_Tank
VAR
	//Tank 1 --- sett global 
	Set_Temp_1: Anaman;
	Tank_Simu_1: Tank_Simulation;
	Tank_Level_1: AnaView;
	Tank_Temp_1: AnaView;
	Tank_Heater_1: binview;

	//Tank 2
	Set_Temp_2: Anaman;
	Tank_Simu_2: Tank_Simulation;
	Tank_Level_2: AnaView;
	Tank_Temp_2: AnaView;
	Tank_Heater_2: binview;

	//Tank 3
	Set_Temp_3: Anaman;
	Tank_Simu_3: Tank_Simulation;
	Tank_Level_3: AnaView;
	Tank_Temp_3: AnaView;
	Tank_Heater_3: binview;

	//Tank 4
	Set_Temp_4: Anaman;
	Tank_Simu_4: Tank_Simulation;
	Tank_Level_4: AnaView;
	Tank_Temp_4: AnaView;
	Tank_Heater_4: binview;
END_VAR

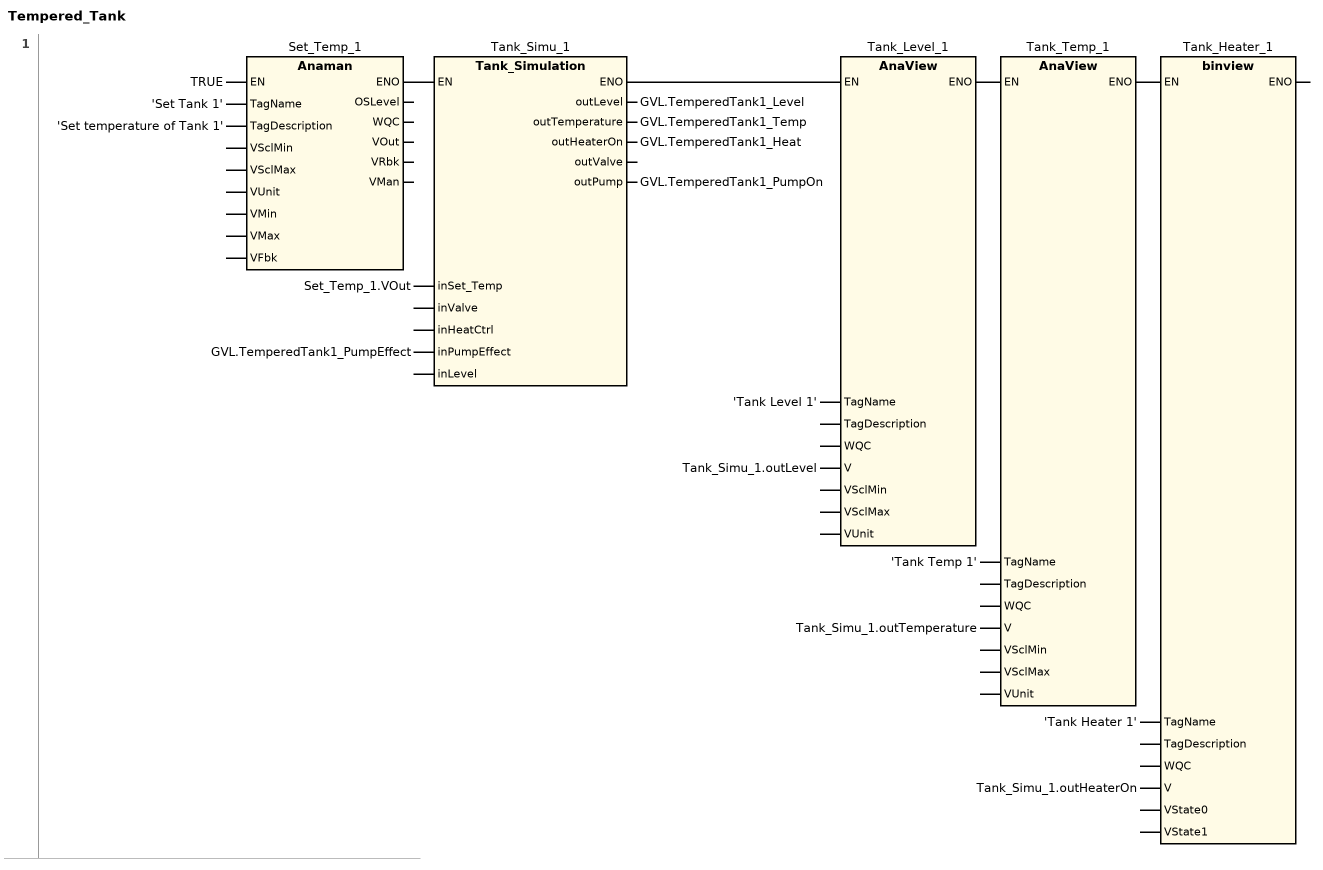
// NETWORK 1
Set_Temp_1(TagName := 'Set Tank 1', TagDescription := 'Set temperature of Tank 1'); // Anaman
Tank_Simu_1(
    inSet_Temp := Set_Temp_1.VOut,
    inPumpEffect := GVL.TemperedTank1_PumpEffect,
    outLevel => GVL.TemperedTank1_Level,
    outTemperature => GVL.TemperedTank1_Temp,
    outHeaterOn => GVL.TemperedTank1_Heat,
    outPump => GVL.TemperedTank1_PumpOn); // Tank_Simulation
Tank_Level_1(TagName := 'Tank Level 1', V := Tank_Simu_1.outLevel); // AnaView
Tank_Temp_1(TagName := 'Tank Temp 1', V := Tank_Simu_1.outTemperature); // AnaView
Tank_Heater_1(TagName := 'Tank Heater 1', V := Tank_Simu_1.outHeaterOn); // binview

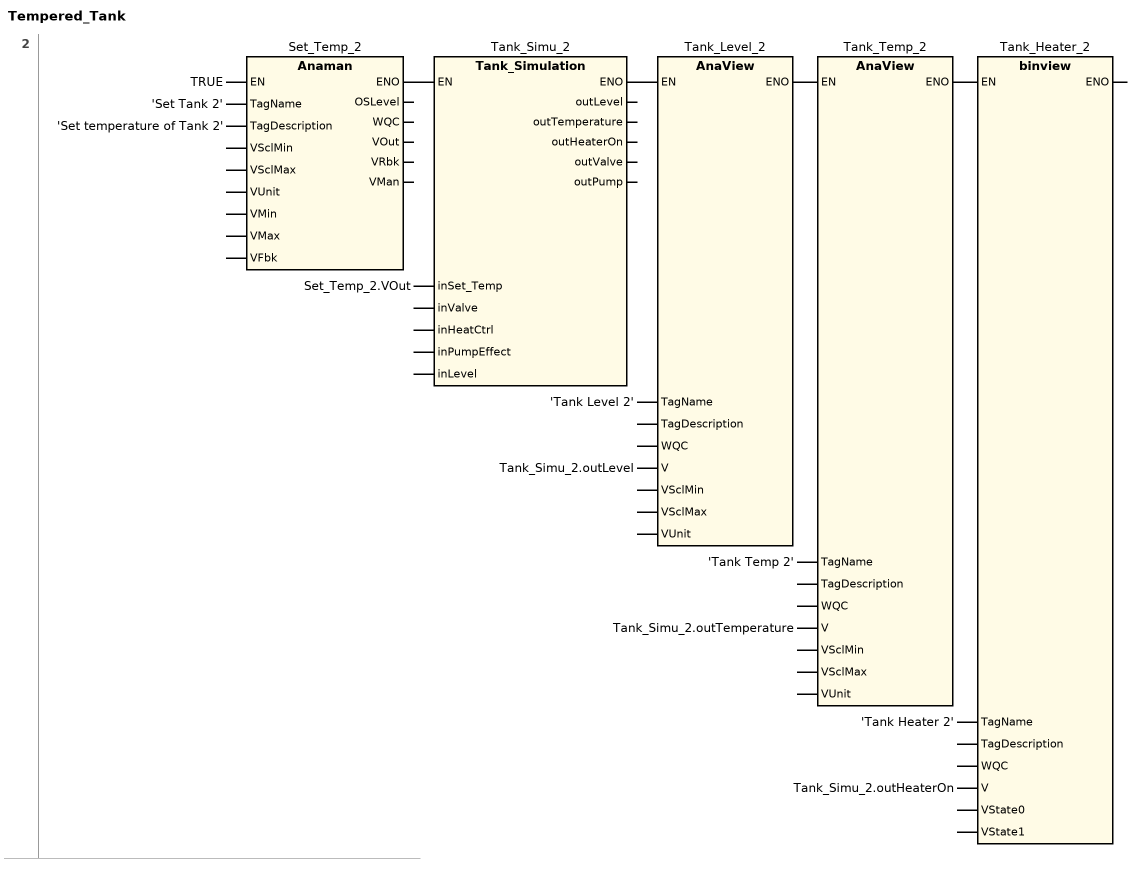
// NETWORK 2
Set_Temp_2(TagName := 'Set Tank 2', TagDescription := 'Set temperature of Tank 2'); // Anaman
Tank_Simu_2(inSet_Temp := Set_Temp_2.VOut); // Tank_Simulation
Tank_Level_2(TagName := 'Tank Level 2', V := Tank_Simu_2.outLevel); // AnaView
Tank_Temp_2(TagName := 'Tank Temp 2', V := Tank_Simu_2.outTemperature); // AnaView
Tank_Heater_2(TagName := 'Tank Heater 2', V := Tank_Simu_2.outHeaterOn); // binview

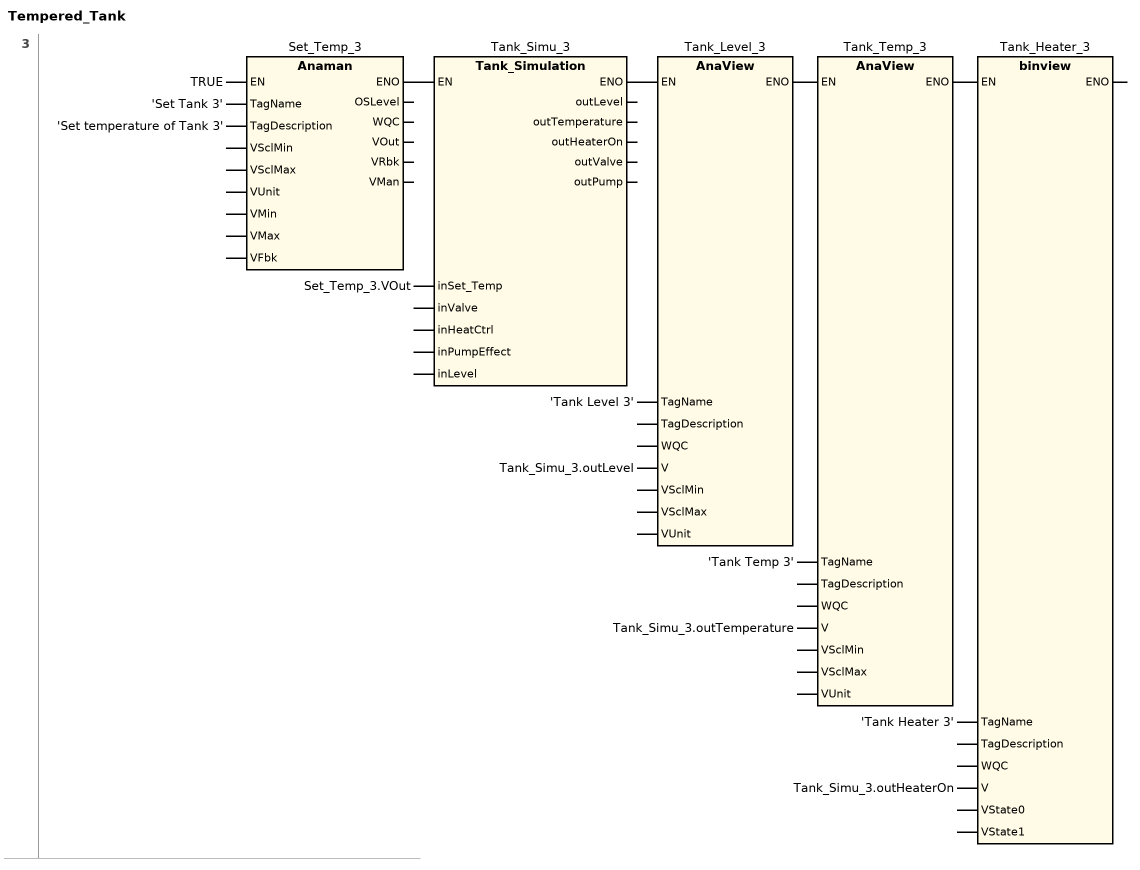
// NETWORK 3
Set_Temp_3(TagName := 'Set Tank 3', TagDescription := 'Set temperature of Tank 3'); // Anaman
Tank_Simu_3(inSet_Temp := Set_Temp_3.VOut); // Tank_Simulation
Tank_Level_3(TagName := 'Tank Level 3', V := Tank_Simu_3.outLevel); // AnaView
Tank_Temp_3(TagName := 'Tank Temp 3', V := Tank_Simu_3.outTemperature); // AnaView
Tank_Heater_3(TagName := 'Tank Heater 3', V := Tank_Simu_3.outHeaterOn); // binview

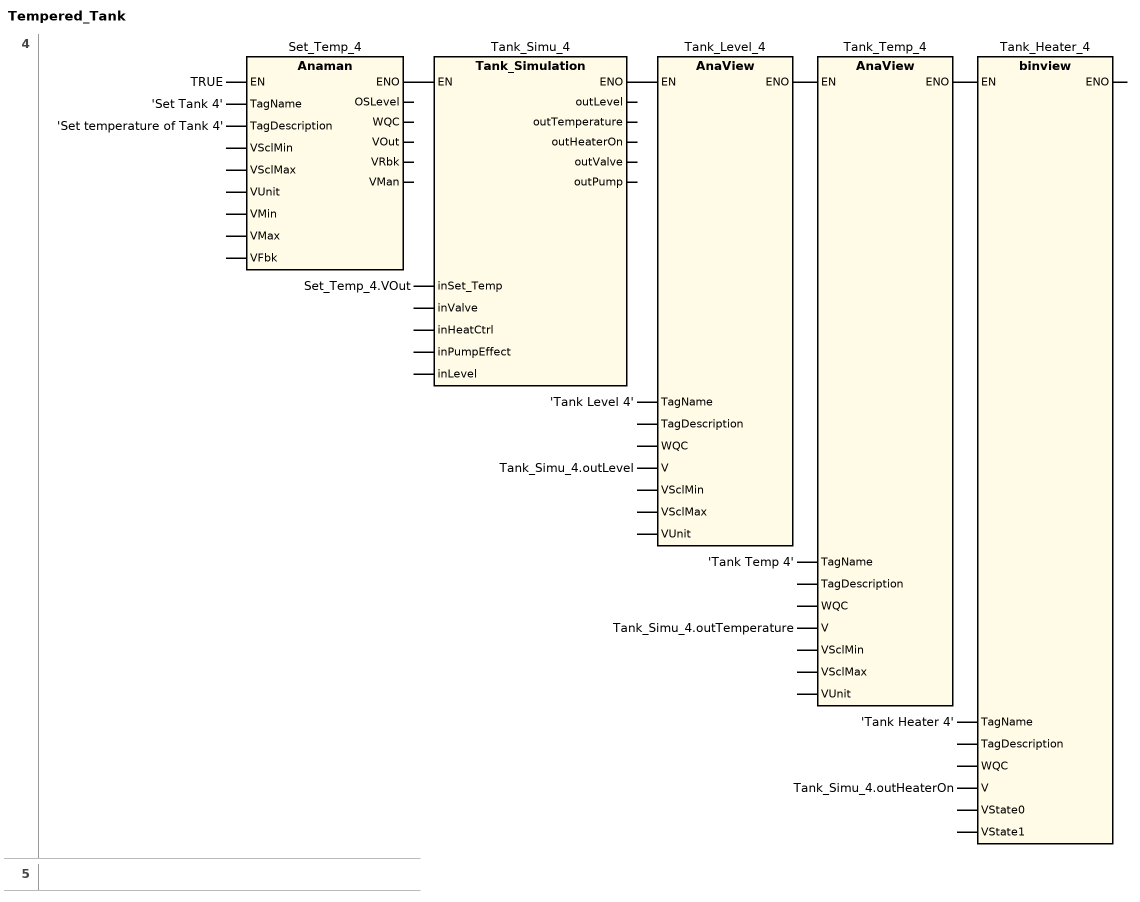
// NETWORK 4
Set_Temp_4(TagName := 'Set Tank 4', TagDescription := 'Set temperature of Tank 4'); // Anaman
Tank_Simu_4(inSet_Temp := Set_Temp_4.VOut); // Tank_Simulation
Tank_Level_4(TagName := 'Tank Level 4', V := Tank_Simu_4.outLevel); // AnaView
Tank_Temp_4(TagName := 'Tank Temp 4', V := Tank_Simu_4.outTemperature); // AnaView
Tank_Heater_4(TagName := 'Tank Heater 4', V := Tank_Simu_4.outHeaterOn); // binview

// NETWORK 5

END_PROGRAM

// Application/Tank_Simulation
FUNCTION_BLOCK Tank_Simulation
VAR_INPUT
	inSet_Temp:	REAL;
	inValve:BOOL;
	inHeatCtrl:BOOL ;
	inPumpEffect:INT;
	inLevel:REAL;
END_VAR
VAR_OUTPUT
	outLevel:	REAL;
	outTemperature:	REAL;
	outHeaterOn:	BOOL;
	outValve:	BOOL;
	outPump	:BOOL;
END_VAR
VAR
	xLevel_Good:BOOL;
	tonTimer:	ton;
	rsTimer:	rs;
	hystHeater: Util.HYSTERESIS;
END_VAR

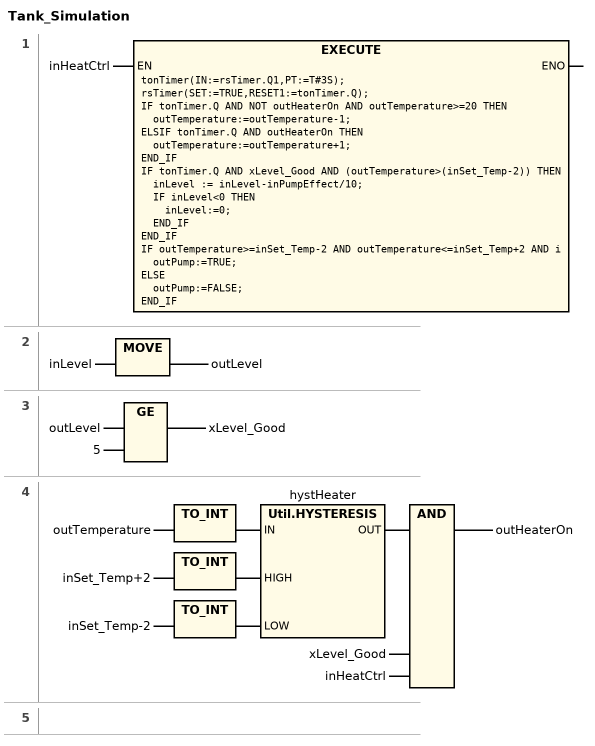
// NETWORK 1
IF inHeatCtrl THEN
    tonTimer(IN:=rsTimer.Q1,PT:=T#3S);
    rsTimer(SET:=TRUE,RESET1:=tonTimer.Q);
    IF tonTimer.Q AND NOT outHeaterOn AND outTemperature>=20 THEN
    	outTemperature:=outTemperature-1;
    ELSIF tonTimer.Q AND outHeaterOn THEN
    	outTemperature:=outTemperature+1;
    END_IF
    IF tonTimer.Q AND xLevel_Good AND (outTemperature>(inSet_Temp-2)) THEN
    	inLevel := inLevel-inPumpEffect/10;
    	IF inLevel<0 THEN 
    		inLevel:=0;
    	END_IF
    END_IF
    IF outTemperature>=inSet_Temp-2 AND outTemperature<=inSet_Temp+2 AND inPumpEffect>0 THEN
    	outPump:=TRUE;
    ELSE
    	outPump:=FALSE;
    END_IF
END_IF

// NETWORK 2
outLevel := inLevel;

// NETWORK 3
xLevel_Good := outLevel >= 5;

// NETWORK 4
hystHeater(IN := TO_INT(outTemperature), HIGH := TO_INT(inSet_Temp+2), LOW := TO_INT(inSet_Temp-2)); // Util.HYSTERESIS
outHeaterOn := hystHeater.OUT AND xLevel_Good AND inHeatCtrl;

// NETWORK 5

END_FUNCTION_BLOCK
